// TIA Portal V18 export
FUNCTION_BLOCK "MixingRatio"   // FB11, LAD
{ S7_Optimized_Access := 'TRUE' }
VERSION : 0.1
// stored: AutoNumber true, IsIECCheckEnabled false, IsRetainMemResEnabled false, MemoryReserve 100, SetENOAutomatically false, UDAEnableTagReadback false
   VAR_INPUT
      "Pump size A in ml" : Real;
      "Pump size B in ml" : Real;
      "Pump speed A_Max" : Real;
      "Pump speed B_Max" : Real;
      "Pump speed A_Passive" : Real;
      "Pump speed B_Passive" : Real;
      "Mixing ratio A100:B" : Real;
      "No.of Component" : Int;
      "Density A" : Real;
      "Density B" : Real;
      "Mixed Flowrate Set" : Real;
      "Flowrate Type" : Int;
   END_VAR
   VAR_OUTPUT
      "Maximum Flowrate A" : Real;
      "Maximum Flowrate B" : Real;
      "Maximum Flowrate A_Limited" : Real;
      "Maximum Flowrate B_Limited" : Real;
      "Maximum Flowrate Mixed" : Real;
      "Required flowrate A" : Real;
      "Required flowrate B" : Real;
   END_VAR
   VAR
      "Pump size A actual" : Real;
      "Pump size B actual" : Real;
      "Max flowrate A" : Real;
      "Max flowrate B" : Real;
      "Ratio margin B" : Real;
      "usable A flowrate per B ratio" : Real;
      "maximum mixed flowrate" : Real;
      "usable flowrate A per ratio" : Real;
      "usable flowrate B per ratio" : Real;
      "Flowrate difference A" : Real;
      "Flowrate difference B" : Real;
      "target flowrate A" : Real;
      "target flowrate B" : Real;
   END_VAR
   VAR_TEMP   // added for the SCL form of the ladder/FBD networks
      _w1 : Bool;
   END_VAR
BEGIN

REGION Network 1
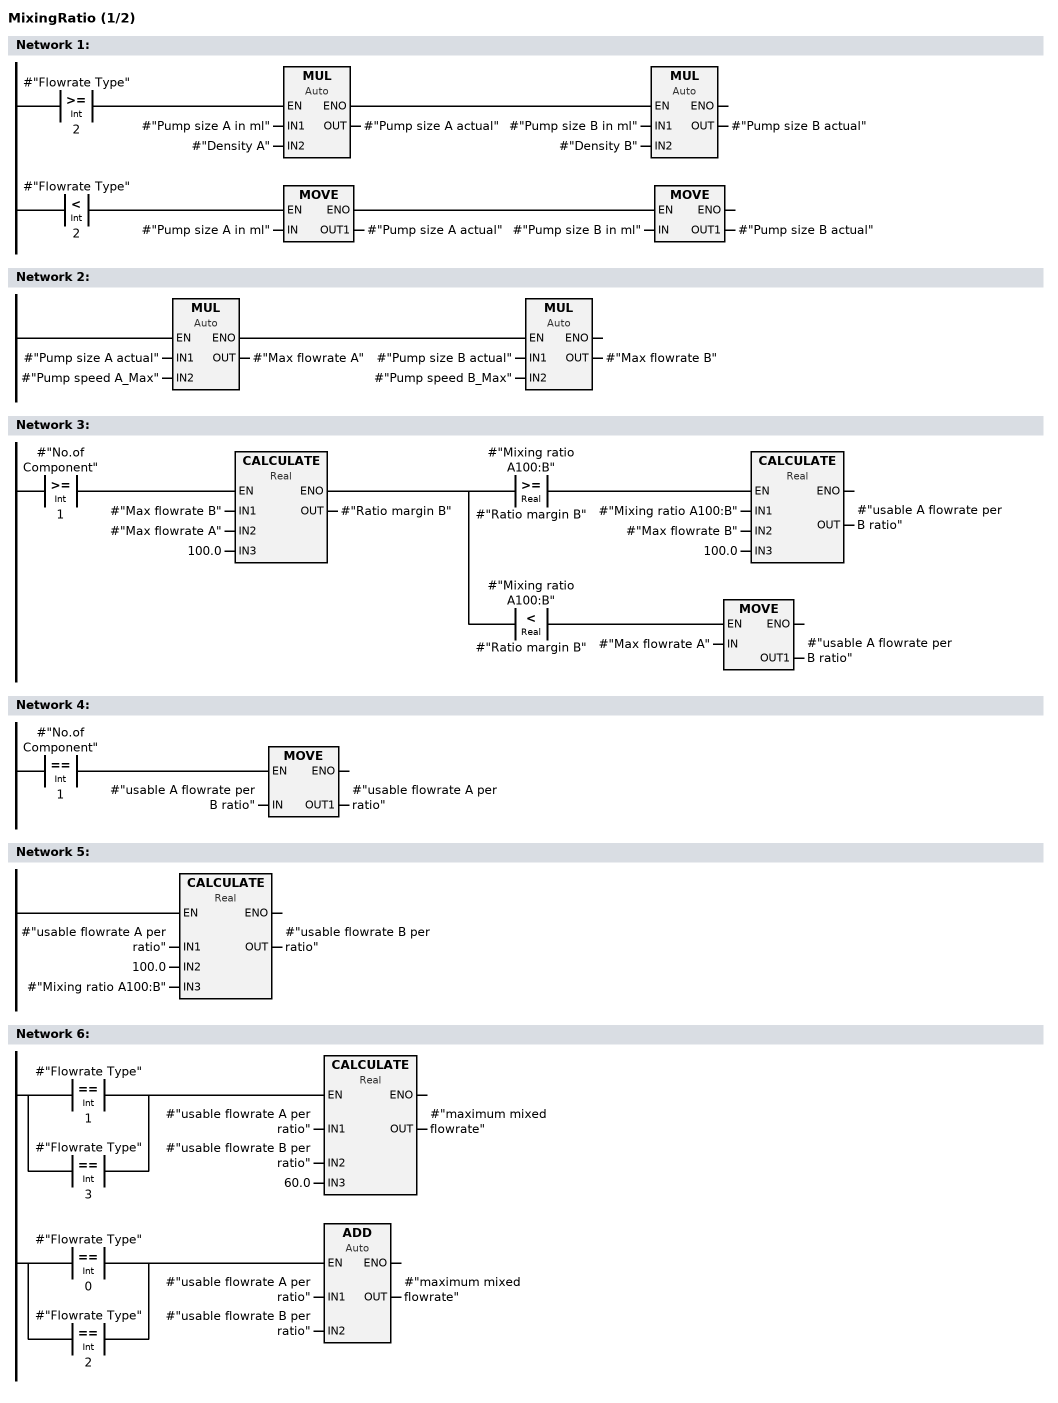
   RUNG wire#powerrail
      { S7_Templates := "SrcType := Int" } GE_Contact(in1 := #"Flowrate Type", in2 := 2)
      Mul(in1 := #"Pump size A in ml", in2 := #"Density A", out => #"Pump size A actual")
      Mul(in1 := #"Pump size B in ml", in2 := #"Density B", out => #"Pump size B actual")
   END_RUNG
   RUNG wire#powerrail
      { S7_Templates := "SrcType := Int" } LT_Contact(in1 := #"Flowrate Type", in2 := 2)
      Move(in := #"Pump size A in ml", out1 => #"Pump size A actual")
      Move(in := #"Pump size B in ml", out1 => #"Pump size B actual")
   END_RUNG
   // the same network as SCL:
   IF #"Flowrate Type" >= 2 THEN
       #"Pump size A actual" := #"Pump size A in ml" * #"Density A";
       #"Pump size B actual" := #"Pump size B in ml" * #"Density B";
   END_IF;
   IF #"Flowrate Type" < 2 THEN
       #"Pump size A actual" := #"Pump size A in ml";
       #"Pump size B actual" := #"Pump size B in ml";
   END_IF;
END_REGION

REGION Network 2
   RUNG wire#powerrail
      Mul(in1 := #"Pump size A actual", in2 := #"Pump speed A_Max", out => #"Max flowrate A")
      Mul(in1 := #"Pump size B actual", in2 := #"Pump speed B_Max", out => #"Max flowrate B")
   END_RUNG
   // the same network as SCL:
   #"Max flowrate A" := #"Pump size A actual" * #"Pump speed A_Max";
   #"Max flowrate B" := #"Pump size B actual" * #"Pump speed B_Max";
END_REGION

REGION Network 3
   RUNG wire#powerrail
      { S7_Templates := "SrcType := Int" } GE_Contact(in1 := #"No.of Component", in2 := 1)
      { S7_Templates := "SrcType := Real"; S7_Expression := "(IN1/IN2)*IN3" } Calculate(in1 := #"Max flowrate B", in2 := #"Max flowrate A", in3 := 100.0, out => #"Ratio margin B")
      wire#w1
      { S7_Templates := "SrcType := Real" } GE_Contact(in1 := #"Mixing ratio A100:B", in2 := #"Ratio margin B")
      { S7_Templates := "SrcType := Real"; S7_Expression := "IN2/(IN1/IN3)" } Calculate(in1 := #"Mixing ratio A100:B", in2 := #"Max flowrate B", in3 := 100.0, out => #"usable A flowrate per B ratio")
   END_RUNG
   RUNG wire#w1
      { S7_Templates := "SrcType := Real" } LT_Contact(in1 := #"Mixing ratio A100:B", in2 := #"Ratio margin B")
      Move(in := #"Max flowrate A", out1 => #"usable A flowrate per B ratio")
   END_RUNG
   // the same network as SCL:
   #_w1 := #"No.of Component" >= 1;
   IF #_w1 THEN #"Ratio margin B" := (#"Max flowrate B"/#"Max flowrate A")*100.0; END_IF;
   IF #_w1 AND (#"Mixing ratio A100:B" >= #"Ratio margin B") THEN
       #"usable A flowrate per B ratio" := #"Max flowrate B"/(#"Mixing ratio A100:B"/100.0);
   END_IF;
   IF #_w1 AND (#"Mixing ratio A100:B" < #"Ratio margin B") THEN
       #"usable A flowrate per B ratio" := #"Max flowrate A";
   END_IF;
END_REGION

REGION Network 4
   RUNG wire#powerrail
      { S7_Templates := "SrcType := Int" } EQ_Contact(in1 := #"No.of Component", in2 := 1)
      Move(in := #"usable A flowrate per B ratio", out1 => #"usable flowrate A per ratio")
   END_RUNG
   // the same network as SCL:
   IF #"No.of Component" = 1 THEN #"usable flowrate A per ratio" := #"usable A flowrate per B ratio"; END_IF;
END_REGION

REGION Network 5
   RUNG wire#powerrail
      { S7_Templates := "SrcType := Real"; S7_Expression := "(IN1/IN2)*IN3" } Calculate(in1 := #"usable flowrate A per ratio", in2 := 100.0, in3 := #"Mixing ratio A100:B", out => #"usable flowrate B per ratio")
   END_RUNG
   // the same network as SCL:
   #"usable flowrate B per ratio" := (#"usable flowrate A per ratio"/100.0)*#"Mixing ratio A100:B";
END_REGION

REGION Network 6
   RUNG wire#powerrail
      { S7_Templates := "SrcType := Int" } EQ_Contact(in1 := #"Flowrate Type", in2 := 1)
      wire#w1
      { S7_Templates := "SrcType := Real"; S7_Expression := "(IN1+IN2)/IN3" } Calculate(in1 := #"usable flowrate A per ratio", in2 := #"usable flowrate B per ratio", in3 := 60.0, out => #"maximum mixed flowrate")
   END_RUNG
   RUNG wire#powerrail
      { S7_Templates := "SrcType := Int" } EQ_Contact(in1 := #"Flowrate Type", in2 := 3)
   END_RUNG wire#w1
   RUNG wire#powerrail
      { S7_Templates := "SrcType := Int" } EQ_Contact(in1 := #"Flowrate Type", in2 := 0)
      wire#w2
      Add(in1 := #"usable flowrate A per ratio", in2 := #"usable flowrate B per ratio", out => #"maximum mixed flowrate")
   END_RUNG
   RUNG wire#powerrail
      { S7_Templates := "SrcType := Int" } EQ_Contact(in1 := #"Flowrate Type", in2 := 2)
   END_RUNG wire#w2
   // the same network as SCL:
   IF (#"Flowrate Type" = 1) OR (#"Flowrate Type" = 3) THEN
       #"maximum mixed flowrate" := (#"usable flowrate A per ratio"+#"usable flowrate B per ratio")/60.0;
   END_IF;
   IF (#"Flowrate Type" = 0) OR (#"Flowrate Type" = 2) THEN
       #"maximum mixed flowrate" := #"usable flowrate A per ratio" + #"usable flowrate B per ratio";
   END_IF;
END_REGION

REGION Network 7
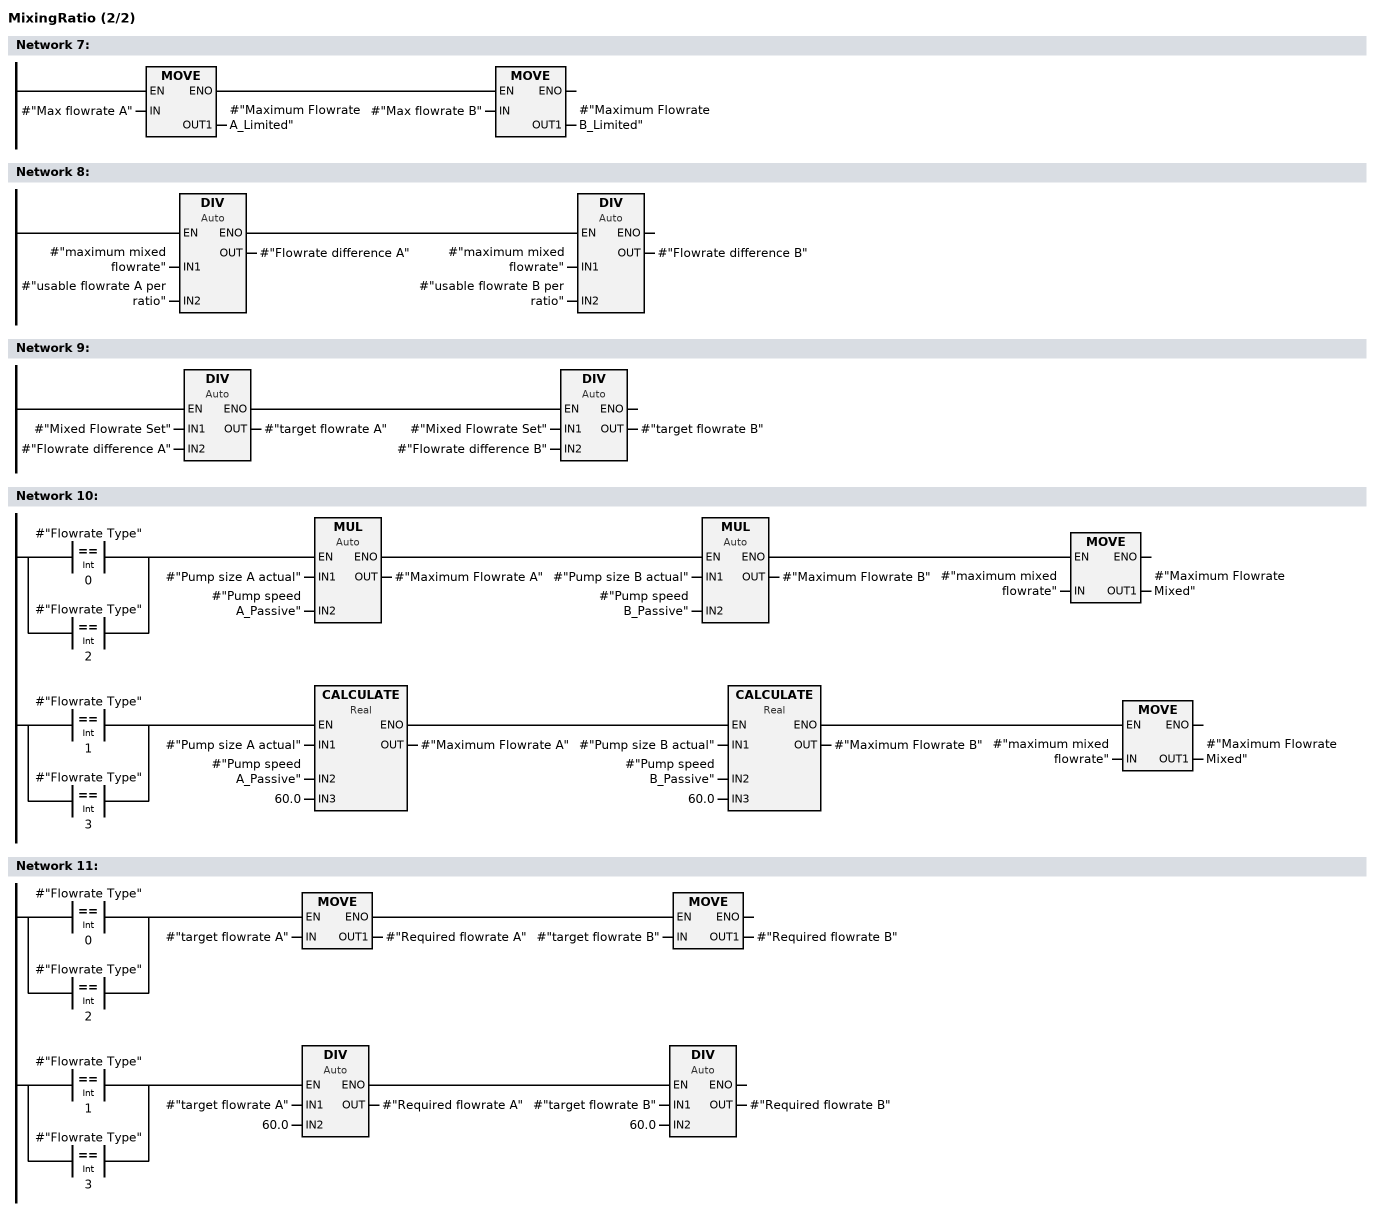
   RUNG wire#powerrail
      Move(in := #"Max flowrate A", out1 => #"Maximum Flowrate A_Limited")
      Move(in := #"Max flowrate B", out1 => #"Maximum Flowrate B_Limited")
   END_RUNG
   // the same network as SCL:
   #"Maximum Flowrate A_Limited" := #"Max flowrate A";
   #"Maximum Flowrate B_Limited" := #"Max flowrate B";
END_REGION

REGION Network 8
   RUNG wire#powerrail
      Div(in1 := #"maximum mixed flowrate", in2 := #"usable flowrate A per ratio", out => #"Flowrate difference A")
      Div(in1 := #"maximum mixed flowrate", in2 := #"usable flowrate B per ratio", out => #"Flowrate difference B")
   END_RUNG
   // the same network as SCL:
   #"Flowrate difference A" := #"maximum mixed flowrate" / #"usable flowrate A per ratio";
   #"Flowrate difference B" := #"maximum mixed flowrate" / #"usable flowrate B per ratio";
END_REGION

REGION Network 9
   RUNG wire#powerrail
      Div(in1 := #"Mixed Flowrate Set", in2 := #"Flowrate difference A", out => #"target flowrate A")
      Div(in1 := #"Mixed Flowrate Set", in2 := #"Flowrate difference B", out => #"target flowrate B")
   END_RUNG
   // the same network as SCL:
   #"target flowrate A" := #"Mixed Flowrate Set" / #"Flowrate difference A";
   #"target flowrate B" := #"Mixed Flowrate Set" / #"Flowrate difference B";
END_REGION

REGION Network 10
   RUNG wire#powerrail
      { S7_Templates := "SrcType := Int" } EQ_Contact(in1 := #"Flowrate Type", in2 := 0)
      wire#w1
      Mul(in1 := #"Pump size A actual", in2 := #"Pump speed A_Passive", out => #"Maximum Flowrate A")
      Mul(in1 := #"Pump size B actual", in2 := #"Pump speed B_Passive", out => #"Maximum Flowrate B")
      Move(in := #"maximum mixed flowrate", out1 => #"Maximum Flowrate Mixed")
   END_RUNG
   RUNG wire#powerrail
      { S7_Templates := "SrcType := Int" } EQ_Contact(in1 := #"Flowrate Type", in2 := 2)
   END_RUNG wire#w1
   RUNG wire#powerrail
      { S7_Templates := "SrcType := Int" } EQ_Contact(in1 := #"Flowrate Type", in2 := 1)
      wire#w2
      { S7_Templates := "SrcType := Real"; S7_Expression := "(IN1*IN2)/IN3" } Calculate(in1 := #"Pump size A actual", in2 := #"Pump speed A_Passive", in3 := 60.0, out => #"Maximum Flowrate A")
      { S7_Templates := "SrcType := Real"; S7_Expression := "(IN1*IN2)/IN3" } Calculate(in1 := #"Pump size B actual", in2 := #"Pump speed B_Passive", in3 := 60.0, out => #"Maximum Flowrate B")
      Move(in := #"maximum mixed flowrate", out1 => #"Maximum Flowrate Mixed")
   END_RUNG
   RUNG wire#powerrail
      { S7_Templates := "SrcType := Int" } EQ_Contact(in1 := #"Flowrate Type", in2 := 3)
   END_RUNG wire#w2
   // the same network as SCL:
   IF (#"Flowrate Type" = 0) OR (#"Flowrate Type" = 2) THEN
       #"Maximum Flowrate A" := #"Pump size A actual" * #"Pump speed A_Passive";
       #"Maximum Flowrate B" := #"Pump size B actual" * #"Pump speed B_Passive";
       #"Maximum Flowrate Mixed" := #"maximum mixed flowrate";
   END_IF;
   IF (#"Flowrate Type" = 1) OR (#"Flowrate Type" = 3) THEN
       #"Maximum Flowrate A" := (#"Pump size A actual"*#"Pump speed A_Passive")/60.0;
       #"Maximum Flowrate B" := (#"Pump size B actual"*#"Pump speed B_Passive")/60.0;
       #"Maximum Flowrate Mixed" := #"maximum mixed flowrate";
   END_IF;
END_REGION

REGION Network 11
   RUNG wire#powerrail
      { S7_Templates := "SrcType := Int" } EQ_Contact(in1 := #"Flowrate Type", in2 := 0)
      wire#w1
      Move(in := #"target flowrate A", out1 => #"Required flowrate A")
      Move(in := #"target flowrate B", out1 => #"Required flowrate B")
   END_RUNG
   RUNG wire#powerrail
      { S7_Templates := "SrcType := Int" } EQ_Contact(in1 := #"Flowrate Type", in2 := 2)
   END_RUNG wire#w1
   RUNG wire#powerrail
      { S7_Templates := "SrcType := Int" } EQ_Contact(in1 := #"Flowrate Type", in2 := 1)
      wire#w2
      Div(in1 := #"target flowrate A", in2 := 60.0, out => #"Required flowrate A")
      Div(in1 := #"target flowrate B", in2 := 60.0, out => #"Required flowrate B")
   END_RUNG
   RUNG wire#powerrail
      { S7_Templates := "SrcType := Int" } EQ_Contact(in1 := #"Flowrate Type", in2 := 3)
   END_RUNG wire#w2
   // the same network as SCL:
   IF (#"Flowrate Type" = 0) OR (#"Flowrate Type" = 2) THEN
       #"Required flowrate A" := #"target flowrate A";
       #"Required flowrate B" := #"target flowrate B";
   END_IF;
   IF (#"Flowrate Type" = 1) OR (#"Flowrate Type" = 3) THEN
       #"Required flowrate A" := #"target flowrate A" / 60.0;
       #"Required flowrate B" := #"target flowrate B" / 60.0;
   END_IF;
END_REGION
END_FUNCTION_BLOCK
